// TIA Portal V20 export
DATA_BLOCK "RealDbName"   // DB7
   VAR
      MyTimer { S7_SetPoint := 'True'} : TON_TIME;
   END_VAR
BEGIN
END_DATA_BLOCK
